Fanuc KAREL source: ka00078.KL

-- PROVISIONAL review KL for V770-1; original PC SHA256 a6bab4a99e9819d60c2c1fb93e52bbb3cb86fd34acd8936423ae53deed5efb40
-- Incomplete behavior may be omitted. Consult companion uncertainty JSON. Do not deploy.
PROGRAM KA00078
%NOLOCKGROUP
-- UNRESOLVED_DECL SRC type=000106
-- UNRESOLVED_DECL DST type=000102
BEGIN
  -- UNRESOLVED_PC offsets 5-20; opcodes 2E,22,32,35
  -- UNRESOLVED_PC offsets 25-45; opcodes 49,7E,4A
  -- UNRESOLVED_PC offsets 50-54; opcodes 7F
END KA00078
